       //disable gas inlet valves 
       //------------------------
       IF (#enb_prs_mon AND ("AV".ACT_PRS_GCH > "CNF".ACC_FNC_PRS_LIM)) THEN
           #dbl_gas_valves    :=  true;
       END_IF;
END_FUNCTION_BLOCK

FUNCTION_BLOCK "BM_MLT_GAP_SEARCH"   // FB117, SCL
{ S7_Optimized_Access := 'FALSE' }
VERSION : 0.0
// --------------------------------------------------------------------------------
//     program     :    BM_MLT_GAP_SEARCH
//     description :    melt gap search
//                          
//     name        :    G. Eibelshaeuser
//     date        :    19.10.2020
// 
//     revision    :
//     name        :
//     date        :    
//                     (c)PVA CGS GmbH
// --------------------------------------------------------------------------------
   VAR
      do_mlt_gap_search : Bool;
      mlt_gap_search_busy : Bool;
      "step" : Int;
      dly : Int;
      start_pos_xt : Real;
      start_pos_cr : Real;
   END_VAR
   VAR CONSTANT
      max_lft_dst : Real := 20.0;   // max lifting distance of crucible or crystal lift in [mm]
   END_VAR
BEGIN


       //disable melt gap search
       //-----------------------
       IF ("STA".ACT_STATE <> "APC".STATE_SERV) OR NOT ("LT".CR_LFT_UP XOR "LT".XT_LFT_DN) OR "LT".LSR_SEN_PWR_ON THEN
           "LT".MLT_GAP_SEARCH   :=  FALSE;
       //enable melt gap search
       //----------------------
       ELSE
           "SM_NEG_EDGE"(input   :=  "KYD".MLT_GAP_SEARCH,
                       busy    :=  #mlt_gap_search_busy,
                       output  :=  "LT".MLT_GAP_SEARCH);
       END_IF;

       //set activation flag melt gap search
       //-----------------------------------
       IF "LT".MLT_GAP_SEARCH THEN
           #do_mlt_gap_search   :=  true;
       END_IF;

       //melt gap search activated
       //-------------------------
       IF #do_mlt_gap_search THEN
           //abort melt gap search
           //---------------------
           IF NOT "LT".MLT_GAP_SEARCH THEN
               #step    :=  50;
           END_IF;

           //sequence
           //--------
           CASE #step OF 

               //switch on melt contact control
               //------------------------------
               0:  "KYD".MCC_ON  :=  TRUE;
                   //set speed set point
                   //-------------------
                   IF "LT".XT_LFT_DN THEN
                       "KYA".SET_XT_SPD  :=  1.0;
                   ELSIF "LT".CR_LFT_UP THEN
                       "KYA".SET_CR_SPD  :=  1.0;
                   END_IF;

                   //activate next step
                   //------------------
                   #step    :=  #step + 10;

               //store start position
               //--------------------
               10: #start_pos_xt    :=  "AV".ACT_XT_POS;
                   #start_pos_cr    :=  "AV".ACT_CR_POS;
                   #dly             :=  0;

                   //activate next step
                   //------------------
                   #step    :=  #step + 10;

               //find contact
               //------------    
               20: //crucible lift moved max. valid distance
                   //---------------------------------------
                   IF ("AV".ACT_CR_POS >= (#start_pos_cr + #max_lft_dst)) THEN
                       "KYD".CR_LFT_OFF          :=  TRUE;
                       "FLT".MLT_GAP_NO_CONTACT  :=  TRUE;
                   //crystal lift moved max. valid distance
                   //-------------------------------------
                   ELSIF ("AV".ACT_XT_POS >= (#start_pos_xt + #max_lft_dst)) THEN
                       "KYD".XT_LFT_OFF          :=  TRUE;
                       "FLT".MLT_GAP_NO_CONTACT  :=  TRUE;
                   //contact detected
                   //----------------
                   ELSIF "PDI".MCC_CONTACT_XT THEN
                       //stop crystal lift
                       //-----------------
                       IF  "LT".XT_LFT_DN THEN
                           "KYD".XT_LFT_OFF  :=  TRUE;
                           //activate next step
                           //------------------
                           #step    :=  #step + 10;
                       //stop crucible lift
                       //-----------------
                       ELSIF  "LT".CR_LFT_UP THEN   
                           "KYD".CR_LFT_OFF  :=  TRUE; 
                           //activate next step
                           //------------------
                           #step    :=  #step + 20;
                       END_IF;
                   END_IF;         

               //crystal - calculate distance
               //----------------------------
               30: IF NOT "LT".XT_LFT_DN THEN
                       //delay next step
                       //---------------
                       IF (#dly > 20) THEN
                           //calculate distance from contact to seed reference position
                           //---------------------------------------------------------- 
                           IF ("DIS".ACT_SEED_LSR_REF_POS > 0.0) THEN
                               "PAR_MAIN".MCONST_DST_LSR_MLT_LVL :=  "AV".ACT_XT_POS - "DIS".ACT_SEED_LSR_REF_POS;
                           END_IF;
                           //activate next step
                           //------------------
                           #step    :=  #step + 20;
                       ELSE
                           IF "SysTick100ms" THEN
                               #dly :=  #dly + 1;
                           END_IF;
                       END_IF;
                   END_IF;

               //crucible - store actual position
               //--------------------------------
               40: IF NOT "LT".CR_LFT_UP THEN
                       //delay next step
                       //---------------
                       IF (#dly > 20) THEN
                           //store actual crucible as dipping position
                           //----------------------------------------- 
                           "DIS".ACT_CR_DIP_POS  := "AV".ACT_CR_POS; 
                           //activate next step
                           //------------------
                           #step    :=  #step + 10;
                       ELSE
                           IF "SysTick100ms" THEN
                               #dly :=  #dly + 1;
                           END_IF;
                       END_IF;
                   END_IF;

               //reset off variables
               //-------------------
               50: "KYD".XT_LFT_OFF      :=  FALSE;
                   "KYD".CR_LFT_OFF      :=  FALSE;
                   "KYA".SET_XT_SPD      :=  0.0;
                   "KYA".SET_CR_SPD      :=  0.0;
                   #do_mlt_gap_search   :=  false;

           END_CASE;

       ELSE
           #step    :=  0;
           "FLT".MLT_GAP_NO_CONTACT  :=  FALSE;
       END_IF;
END_FUNCTION_BLOCK

FUNCTION_BLOCK "BM_SEED_REF_POS"   // FB118, SCL
{ S7_Optimized_Access := 'FALSE' }
VERSION : 0.0
// --------------------------------------------------------------------------------
//     program     :    BM_SEED_REF_POS
//     description :    seed reference position search
//                          
//     name        :    G. Eibelshaeuser
//     date        :    18.12.2020
// 
//     revision    :
//     name        :
//     date        :    
//                     (c)PVA CGS GmbH
// --------------------------------------------------------------------------------
   VAR
      do_ref_search : Bool;
      seed_search_busy : Bool;
      lsr_sen_obj_det : Bool;
      "step" : Int;
      dly : Int;
      start_pos_xt : Real;
   END_VAR
   VAR CONSTANT
      max_lft_dst : Real := 20.0;   // max lifting distance of crucible or crystal lift in [mm]
   END_VAR
BEGIN


       //switch on laser in dipping phase
       //--------------------------------
       IF ("APC".STATUS = "APC".DIPPING) THEN
           "LT".LSR_SEN_PWR_ON   :=  TRUE;        
       //disable reference search
       //------------------------
       ELSIF "APC".AUTOMATIC OR NOT "LT".XT_LFT_DN OR "LT".MLT_GAP_SEARCH THEN
           "LT".LSR_SEN_PWR_ON   :=  FALSE;
       //enablereference search
       //----------------------
       ELSE
           "SM_NEG_EDGE"(input   :=  "KYD".LSR_SEN_PWR_ON,
                       busy    :=  #seed_search_busy,
                       output  :=  "LT".LSR_SEN_PWR_ON);
       END_IF;

       //set activation flag melt gap search
       //-----------------------------------
       IF ("LT".LSR_SEN_PWR_ON AND ("APC".STATUS = "APC".IDLE))THEN
           #do_ref_search   :=  true;
       END_IF;

       //reference search activated
       //--------------------------
       IF #do_ref_search THEN
           //abort reference position search
           //-------------------------------
           IF (NOT "LT".LSR_SEN_PWR_ON AND (#step < 25)) THEN
               #step    :=  40;
           END_IF;

           //sequence
           //--------
           CASE #step OF 
               //switch on melt contact control
               //------------------------------
               0:  //set speed set point
                   //-------------------
                   "KYA".SET_XT_SPD              :=  1.0;
                   "DIS".ACT_SEED_LSR_REF_POS    :=  0.0;
                   #dly                         :=  0;
                   //activate next step
                   //------------------
                   #step    :=  #step + 10;

               //store start position
               //--------------------
               10: #start_pos_xt    :=  "AV".ACT_XT_POS;
                   //activate next step
                   //------------------
                   #step    :=  #step + 10;

               //find contact
               //------------    
               20: //crystal lift moved max. valid distance
                   //-------------------------------------
                   IF ("AV".ACT_XT_POS >= (#start_pos_xt + #max_lft_dst)) THEN
                       "KYD".XT_LFT_OFF  :=  TRUE;
                       //activate next step
                       //------------------
                       #step    :=  #step + 5;
                   //reference position detected with positive edge of laser sensor
                   //--------------------------------------------------------------
                   ELSIF ("PDI".LSR_SEN_OBJ_DET AND NOT #lsr_sen_obj_det) THEN
                       "KYD".XT_LFT_OFF  :=  TRUE;
                       //activate next step
                       //------------------
                       #step    :=  #step + 10;
                   END_IF;

               25: //crystal lift stopped - no seed detected within valid range
                   //----------------------------------------------------------
                   IF NOT "LT".XT_LFT_DN THEN
                       "FLT".SEED_DET    :=  TRUE;
                       //delay next step
                       //---------------
                       IF (#dly > 20) THEN 
                           //activate next step
                           //------------------
                           #step    :=  #step + 15;
                       ELSE
                           IF "SysTick100ms" THEN
                               #dly :=  #dly + 1;
                           END_IF;
                       END_IF;
                   END_IF;

               30: //crystal lift stopped - position stored
                   //--------------------------------------
                   IF NOT "LT".XT_LFT_DN THEN
                       //delay next step
                       //---------------
                       IF (#dly > 20) THEN 
                           //store actual position as reference position
                           //-------------------------------------------
                           "DIS".ACT_SEED_LSR_REF_POS    :=  "AV".ACT_XT_POS;
                           //activate next step
                           //------------------
                           #step    :=  #step + 10;
                       ELSE
                           IF "SysTick100ms" THEN
                               #dly :=  #dly + 1;
                           END_IF;
                       END_IF;

                   END_IF;

               //reset off variables
               //-------------------
               40: "KYD".XT_LFT_OFF      :=  FALSE;
                   "KYA".SET_XT_SPD      :=  0.0;
                   "LT".LSR_SEN_PWR_ON   :=  FALSE;
                   #do_ref_search       :=  false;

           END_CASE;

       ELSE
           #step            :=  0;
           "FLT".SEED_DET    :=  FALSE;
       END_IF;

       //store status of current cycle
       //-----------------------------
       #lsr_sen_obj_det :=  "PDI".LSR_SEN_OBJ_DET;

       //set output laser power on
       //-------------------------
       "PDO".LSR_SEN_PWR_ON  :=  NOT "LT".LSR_SEN_PWR_ON;  //output must be "false" for laser on!!!
END_FUNCTION_BLOCK

FUNCTION_BLOCK "CM_PT1"   // FB130, SCL
{ S7_Optimized_Access := 'FALSE' }
VERSION : 0.0
// --------------------------------------------------------------------------------
//     program     :    CM_PT1
//     description :    pt1 filter 
//     name        :    K. Kalkowski
//     date        :    29.10.99
// 
//     revision    :    1.00
//     name        :    K. Kalkowski
//     date        :    29.10.99
// 
//                     (c)LEYBOLD SYSTEMS
//     --------------------------------------------------------------------------------
   VAR_INPUT
      u_in : Real;   // filter input
      t1_in : Real;   // filter time in sec.
      ts_in : Real;   // filter sample time
      tc_in : Real;   // interrupt time for filter module call (ts/tc>=1, ts/tc=integer!)
      range_in : Real;   // value for 100% input (e.g. 8mm/min = 100%) used for u_in
      range_out : Real;   // value for 100% output (e.g. 700C = 100%) used for y_out
      y_llim : Real;   // low limit for y_out
      y_hlim : Real;   // high limit for y_out
   END_VAR
   VAR_IN_OUT
      y_out : Real;   // pt1 filter output
   END_VAR
   VAR
      u : Real;   // filter input
      y_sum : Real;   // sum of pt1 components
      filter_call_cycle : Int;   // pt1 algorithm call every (ts/tc) cycles
      hlim_active : Bool;   // hlim active
      llim_active : Bool;   // llim active
      filter_off : Bool;   // filter function off (T1 = 0)
      ctrl_call_cycle : Int;   // pt1 algorithm call every (ts/tc) cycles
   END_VAR
BEGIN


       IF #range_in = 0 THEN                                            //check range_in value
           #u:= 0;
       ELSE
           #u:= #u_in / #range_in;
       END_IF;

       IF  #ctrl_call_cycle >= REAL_TO_INT(#ts_in/#tc_in)THEN             //wait for next controller call                               
           #ctrl_call_cycle := 1;
           IF #t1_in <= 0.0 THEN
               #filter_off := true;      
           ELSE
               #filter_off := false;      
           END_IF;
           IF #filter_off = false THEN
               ENO:=TRUE;
               #y_sum := #y_sum + (#u - #y_sum) * (#ts_in/#t1_in);           //calculate filter function
               IF ENO = FALSE THEN
                   #y_sum:=0.0;
               END_IF; 
           ELSE
               #y_sum := #u;
           END_IF;
       ELSE    
           #ctrl_call_cycle := #ctrl_call_cycle + 1;
       END_IF;

       IF #y_sum > #y_hlim / #range_out THEN                              //limit and convert output
           #y_sum := #y_hlim / #range_out;
           #hlim_active := true;
       ELSE
           #hlim_active := false;
       END_IF;
       IF #y_sum < #y_llim / #range_out THEN
           #y_sum := #y_llim / #range_out;
           #llim_active := true;     
       ELSE
           #llim_active := false;
       END_IF;                                                              
       #y_out := #y_sum * #range_out;                                     //set output value
END_FUNCTION_BLOCK

FUNCTION_BLOCK "CM_PT2"   // FB131, SCL
{ S7_Optimized_Access := 'FALSE' }
VERSION : 0.0
// --------------------------------------------------------------------------------
//     program     :    CM_PT2
//     description :    pt2 filter 
//     name        :    G. Eibelsh鋟ser
//     date        :    20.02.2001
// 
//     revision    :    
//     name        :    
//     date        :    
// 
//                     (c)CGS
//     --------------------------------------------------------------------------------
   VAR_INPUT
      u_in : Real;   // filter input
      t1_in : Real;   // filter time 1 in sec.
      t2_in : Real;   // filter time 2 in sec.
      ts_in : Real;   // filter sample time
      tc_in : Real;   // interrupt time for filter module call (ts/tc>=1, ts/tc=integer!)
      range_in : Real;   // value for 100% input (e.g. 8mm/min = 100%) used for u_in
      range_out : Real;   // value for 100% output (e.g. 700C = 100%) used for y_out
      y_llim : Real;   // low limit for y_out
      y_hlim : Real;   // high limit for y_out
   END_VAR
   VAR_IN_OUT
      y_out : Real;   // pt2 filter output
   END_VAR
   VAR
      u : Real;   // filter input
      y_sum : Real;   // sum of pt2 components
      filter_call_cycle : Int;   // pt2 algorithm call every (ts/tc) cycles
      hlim_active : Bool;   // hlim active
      llim_active : Bool;   // llim active
      filter_off : Bool;   // filter function off (T1 = 0)
      ctrl_call_cycle : Int;   // pt2 algorithm call every (ts/tc) cycles
   END_VAR
BEGIN


       IF #range_in = 0 THEN                                            //check range_in value
           #u:= 0;
       ELSE
           #u:= #u_in / #range_in;
       END_IF;

       IF  #ctrl_call_cycle >= REAL_TO_INT(#ts_in/#tc_in)THEN             //wait for next controller call                               
           #ctrl_call_cycle := 1;

           IF (#t1_in <= 0.0)  THEN
               #filter_off := true;      
           ELSE
               #filter_off := false;      
           END_IF;

           IF #filter_off = false THEN
               ENO:= TRUE;
               #y_sum := #y_sum + (#u - #y_sum) * #ts_in/(1+#t1_in+#t2_in+#t1_in*#t2_in);   //calculate filter function
               IF ENO = FALSE THEN
                   #y_sum:=0.0;
               END_IF; 
           ELSE
               #y_sum := #u;
           END_IF;
       ELSE    
           #ctrl_call_cycle := #ctrl_call_cycle + 1;
       END_IF;

       IF #y_sum > #y_hlim / #range_out THEN                              //limit and convert output
           #y_sum := #y_hlim / #range_out;
           #hlim_active := true;
       ELSE
           #hlim_active := false;
       END_IF;
       IF #y_sum < #y_llim / #range_out THEN
           #y_sum := #y_llim / #range_out;
           #llim_active := true;     
       ELSE
           #llim_active := false;
       END_IF;                                                              
       #y_out := #y_sum * #range_out;                                     //set output value
END_FUNCTION_BLOCK

FUNCTION_BLOCK "CM_DT1"   // FB132, SCL
{ S7_Optimized_Access := 'FALSE' }
VERSION : 0.0
// --------------------------------------------------------------------------------
//     program     :    CM_DT1
//     description :    dt1 derivative function with delay 
//     name        :    K. Kalkowski
//     date        :    26.11.99
// 
//     revision    :    1.00
//     name        :    K. Kalkowski
//     date        :    26.11.99
// 
//                     (c)LEYBOLD SYSTEMS
//     --------------------------------------------------------------------------------
   VAR_INPUT
      u_in : Real;   // function input
      td_in : Real;   // derivative time const. in sec.
      t1_in : Real;   // derivative delay time in sec.
      ts_in : Real;   // function sample time
      tc_in : Real;   // interrupt time for function module call (ts/tc>=1, ts/tc=integer!)
      range_in : Real;   // value for 100% input (e.g. 8mm/min = 100%) used for u_in
      range_out : Real;   // value for 100% output (e.g. 700C = 100%) used for y_out
      y_llim : Real;   // low limit for y_out
      y_hlim : Real;   // high limit for y_out
   END_VAR
   VAR_IN_OUT
      y_out : Real;   // dt1 function output
   END_VAR
   VAR
      u : Real;   // function input
      u_old : Real;   // previous of u
      y_sum : Real;   // sum of dt1 components
      funct_call_cycle : Int;   // dt1 algorithm call every (ts/tc) cycles
      hlim_active : Bool;   // hlim active
      llim_active : Bool;   // llim active
      funct_off : Bool;   // dt1 function off (Td = 0)
      ctrl_call_cycle : Int;   // dt1 algorithm call every (ts/tc) cycles
      xd : Real;   // set - act
      xd_old : Real;   // previous value of xd
      du : Real;   // u - u_old
      dxr : Real;   // xr n (differenzenquotient)
      dxr_old : Real;   // xr,n-1 (previous differenzenquotient)
   END_VAR
BEGIN


       IF #range_in = 0 THEN                                        //check range_in value
           #u:= 0;
       ELSE
           #u:= #u_in / #range_in;
           //dxr := 0;
       END_IF;

       IF  #ctrl_call_cycle >= REAL_TO_INT(#ts_in/#tc_in)THEN         //wait for next controller call                               
           #ctrl_call_cycle := 1;
           #du := #u - #u_old;                                        //calculate input                                         
           IF #td_in <= 0.0 THEN
               #funct_off := true;      
           ELSE
               #funct_off := false;      
           END_IF;
           IF #funct_off = false THEN                               //calculate dt1 function
               ENO:=TRUE;
               #dxr := (#du + (#t1_in * #dxr_old)) / (#ts_in + #t1_in);  //differenzenquotient
               IF ENO = FALSE THEN
                   #dxr_old:=0.0;
                   #dxr:=0.0;
               END_IF;              
               #y_sum := #td_in * #dxr;                               //dt1    
           ELSE
               #y_sum := #u;
           END_IF;
           #u_old := #u;                                                 //save previous values
           #dxr_old := #dxr;
       ELSE    
           #ctrl_call_cycle := #ctrl_call_cycle + 1;
       END_IF;

       IF #y_sum > #y_hlim / #range_out THEN                          //limit and convert output
           #y_sum := #y_hlim / #range_out;
           #hlim_active := true;
       ELSE
           #hlim_active := false;
       END_IF;
       IF #y_sum < #y_llim / #range_out THEN
           #y_sum := #y_llim / #range_out;
           #llim_active := true;     
       ELSE
           #llim_active := false;
       END_IF;                                                              
       #y_out := #y_sum * #range_out;                                 //set output value
END_FUNCTION_BLOCK

FUNCTION_BLOCK "CM_INC"   // FB133, SCL
{ S7_Optimized_Access := 'FALSE' }
VERSION : 0.0
// --------------------------------------------------------------------------------
//     program     :    CM_INC
//     description :    increment function  
//     name        :    K. Kalkowski
//     date        :    26.11.99
// 
//     revision    :    1.00
//     name        :    K. Kalkowski
//     date        :    26.11.99
//     
//     revision    :    minimum increment limit added
//     name        :    G. Eibelsh鋟ser
//     date        :    28.11.2011
// 
//                     (c)PVA TePla AG
//     --------------------------------------------------------------------------------
   VAR_INPUT
      u1_in : Real;   // increment input 1
      u2_in : Real;   // increment input 2
      u3_in : Real;   // increment input 3
      k1_in : Real;   // factor for increment input 1
      k2_in : Real;   // factor for increment input 2
      k3_in : Real;   // factor for increment input 3
      y0_in : Real;   // start value input
      y_llim : Real;   // low limit for y_out
      y_hlim : Real;   // high limit for y_out
      y0_mode : Bool;   // set start value of increment function
   END_VAR
   VAR_IN_OUT
      y_out : Real;   // inc function output
      stp_1 : Bool;   // stop increment function (used for change of input connection)
      stp_2 : Bool;
      stp_3 : Bool;
      rstrt_1 : Bool;   // restart increment function (used for start of new increment table)
      rstrt_2 : Bool;
      rstrt_3 : Bool;
   END_VAR
   VAR
      u1_old : Real;   // increment 1 input of previous call
      u2_old : Real;   // increment 2 input of previous call
      u3_old : Real;   // increment 3 input of previous call
      y0 : Real;   // start value
      y_sum : Real;   // sum of increments
      stp1_i : Int;   // index stop function
      stp2_i : Int;
      stp3_i : Int;
      rstrt1_i : Int;   // index restart function
      rstrt2_i : Int;
      rstrt3_i : Int;
   END_VAR
   VAR CONSTANT
      min_inc : Real := 0.001;
   END_VAR
BEGIN


       IF #stp_1 THEN                                    //stop inc function
           #stp1_i := #stp1_i + 1;
           IF (#stp1_i > 2) THEN
               #stp_1 := false;
           END_IF;    
       ELSE
           #stp1_i := 0;
       END_IF;    

       IF #stp_2 THEN
           #stp2_i := #stp2_i + 1;
           IF (#stp2_i > 2) THEN
               #stp_2 := false;
           END_IF;    
       ELSE
           #stp2_i := 0;
       END_IF;    

       IF #stp_3 THEN
           #stp3_i := #stp3_i + 1;
           IF (#stp3_i > 2) THEN
               #stp_3 := false;
           END_IF;    
       ELSE
           #stp3_i := 0;
       END_IF;    

       IF #rstrt_1 THEN                                  //restart inc function
           #rstrt1_i := #rstrt1_i + 1;
           IF (#rstrt1_i > 2) THEN
               #rstrt_1 := false;
           END_IF;    
       ELSE
           #rstrt1_i := 0;
       END_IF;    

       IF #rstrt_2 THEN                                    
           #rstrt2_i := #rstrt2_i + 1;
           IF (#rstrt2_i > 2) THEN
               #rstrt_2 := false;
           END_IF;    
       ELSE
           #rstrt2_i := 0;
       END_IF;    

       IF #rstrt_3 THEN                                    
           #rstrt3_i := #rstrt3_i + 1;
           IF (#rstrt3_i > 2) THEN
               #rstrt_3 := false;
           END_IF;    
       ELSE
           #rstrt3_i := 0;
       END_IF;    

       IF NOT #y0_mode THEN                                         //calculate y_sum
           IF NOT (#rstrt_1 OR #stp_1) THEN 
               IF (ABS(#u1_in - #u1_old) >= #min_inc) THEN            //check if increment is larger than minimum increment limit           
                   #y_sum   := #y_sum + ((#u1_in - #u1_old)*#k1_in);
                   #u1_old  := #u1_in;                               //store last input value
               END_IF;
           END_IF;

           IF NOT (#rstrt_2 OR #stp_2) THEN
               IF (ABS(#u2_in - #u2_old) >= #min_inc) THEN                  
                   #y_sum   := #y_sum + ((#u2_in - #u2_old)*#k2_in);
                   #u2_old  := #u2_in;
               END_IF;
           END_IF;

           IF NOT (#rstrt_3 OR #stp_3) THEN
               IF (ABS(#u3_in - #u3_old) >= #min_inc) THEN                  
                   #y_sum   := #y_sum + ((#u3_in - #u3_old)*#k3_in);
                   #u3_old  := #u3_in;
               END_IF;
           END_IF;

       ELSE
           #y_sum   := #y0_in;
           #u1_old  := #u1_in;
           #u2_old  := #u2_in;
           #u3_old  := #u3_in;

       END_IF;

       IF #y_sum > #y_hlim THEN                                  //limit y_sum
           #y_sum := #y_hlim;    
       END_IF;
       IF #y_sum < #y_llim THEN
           #y_sum := #y_llim;    
       END_IF;

       IF #rstrt_1 THEN                                         //reset previous values
           #u1_old := 0.0;
       END_IF;

       IF #stp_1 THEN
           #u1_old := #u1_in;
       END_IF;

       IF #rstrt_2 THEN
           #u2_old := 0.0;
       END_IF;

       IF #stp_2 THEN
           #u2_old := #u2_in;
       END_IF;

       IF #rstrt_3 THEN
           #u3_old := 0.0;
       END_IF;

       IF #stp_3 THEN
           #u3_old := #u3_in;
       END_IF;

       #y_out := #y_sum;                                         //set output
END_FUNCTION_BLOCK

FUNCTION_BLOCK "CM_LOOP_PRS"   // FB134, SCL
{ S7_Optimized_Access := 'FALSE' }
VERSION : 0.0
// --------------------------------------------------------------------------------
//     program     :    CM_LOOP_PRS
//     description :    pressure control loop 
//     name        :    K. Kalkowski
//     date        :    07.12.99
// 
//     revision    :    call of CONT_C added as alternative
//     name        :    G. Eibelsh鋟ser
//     date        :    06.09.2007
//    
//     revision    :    
//     name        :    
//     date        :    
// 
//                     (c)PVA TePla AG
//     --------------------------------------------------------------------------------
   VAR
      STD_PID : CONT_C;   // standard Siemens controller algorithm
      PT1 : "CM_PT1";   // pt1 filter for actual xtal diameter
      ramp_enb : Bool;
      cyc_cnt : Bool;
      int_hold_req : Bool;   // integral hold action request
      ctl_prs_on : Bool;
      cycle : Int;
      count : Int;
      ctrl_calls : Int;   // controller call counter
      set : Real;   // internal set point
      act : Real;   // internal actual value
      hand : Real;   // internal hand value
      set_ramp : Real;
   END_VAR
   VAR_TEMP
      high_lim_active : Bool;   // high limit of controller output is reached
      low_lim_active : Bool;   // low limit of controller output is reached
      int_action_on : Bool;   // integral action on
      der_action_on : Bool;   // derivative action on
      per_out : Word;   // peripherial controller output variable
      p_part_out : Real;   // proportionality component
      i_part_out : Real;   // integral component
      d_part_out : Real;   // derivative component
      eff_act_val : Real;   // effective process variable
      error_sig : Real;   // control deviation
   END_VAR
   VAR CONSTANT
      nc : Real := 0.0;   // "not connected input"
   END_VAR
BEGIN


       //build hand value
       //---------------- 
       #hand := "CM_INSELECT" (auto   := ("APC".AUTOMATIC AND NOT "SY".CTL_PRS_SMI) OR "DV".SI_FIL_FSH_SEQ_ON,        
                            track  := false,
                            ac     := "AC".SET_CTL_VALVE_POS,                
                            kya    := "KYA".SET_CTL_VALVE_POS);                    

       //build set point
       //---------------
       #set := "CM_INSELECT"(auto    := "APC".AUTOMATIC AND NOT "SY".CTL_PRS_SMI,            
                          track   := true,
                          ac      := "AC".SET_CLF_PRS,
                          kya     := "KYA".SET_PRS_FNC);

       //limitation of pressure control setpoint if no 1000mbar Baratron on furnace chamber present
       //-----------------------------------------------------------------------------------------                   
       IF NOT "CNF".CONF_CLF_BAR_1000    THEN        // check config flag
           IF #set > 90.0 THEN                      // pressure control setpoint limited to 90 mbar
               #set             := 90.0;
               "KYA".SET_PRS_FNC := #set;       
           END_IF;
       END_IF;                    

       #act := "AV".ACT_PRS_FCH;                              //read actual value

       //built controller on flag
       //------------------------
       IF "DV".SI_FIL_FSH_SEQ_ON OR NOT "PDI".EMO THEN 
           "SY".CTL_PRS_ON := FALSE;                 
       ELSIF "DV".FIL_CLN_REQ_IN_PRC THEN        //prevent switch off of pressure control when filter cleaning during process is active
           "SY".CTL_PRS_ON := TRUE;                 
       ELSIF "APC".AUTOMATIC THEN  
           "SY".CTL_PRS_ON := "DC".CTL_PRS_ON;                 
       ELSE 
           "SY".CTL_PRS_ON := ("SY".CTL_PRS_ON AND NOT "KYD".CTL_PRS_OFF) OR "KYD".CTL_PRS_ON; 
       END_IF;

       //setpoint ramping
       //----------------
       IF "SY".CTL_PRS_ON    THEN
           // call setpoint ramp function after controller start
           //---------------------------------------------------
           IF ("PAR_SUB".PRS_RP_GRAD > 0.0)     THEN
               "CM_SET_RAMP"(rp_enb      := #ramp_enb,
                           i           := #cyc_cnt,
                           max_dev     := "PAR_SUB".PRS_RP_MAX_DEV,
                           rp_start    := "PAR_SUB".PRS_RP_START,
                           rp_grad     := "PAR_SUB".PRS_RP_GRAD,
                           tme_base    := 60.0,
                           tc_in       := 0.1,
                           set_p       := #set,
                           act_v       := #act,
                           set_out     := #set_ramp);

               #set     := #set_ramp; 
           END_IF;  
       ELSE
           #ramp_enb  := TRUE;     
           #cyc_cnt   := TRUE;                
       END_IF;

       //write setpoint in KYA variable 
       //------------------------------
       IF "APC".AUTOMATIC AND NOT "SY".CTL_PRS_SMI THEN   
           "KYA".SET_PRS_FNC := #set;
       END_IF;

       "LT".CTL_PRS_ON := "SY".CTL_PRS_ON;                             

       //chose parameter set according to pressure setpoint
       //--------------------------------------------------
       IF #set <= 100.0 THEN
           "AC".CTL_PRS_GN := "PAR_MAIN".CTL_PRS_GN;               //fetch pid parameter from par_main db
           "AC".CTL_PRS_TI := "PAR_MAIN".CTL_PRS_TI;
           "AC".CTL_PRS_TD := "PAR_MAIN".CTL_PRS_TD;
           "AC".CTL_PRS_T1 := "PAR_MAIN".CTL_PRS_T1;    
       ELSE
           "AC".CTL_PRS_GN := "PAR_MAIN".CTL_PRS_GN_HI;               //fetch pid parameter from par_main db
           "AC".CTL_PRS_TI := "PAR_MAIN".CTL_PRS_TI_HI;
           "AC".CTL_PRS_TD := "PAR_MAIN".CTL_PRS_TD_HI;
           "AC".CTL_PRS_T1 := "PAR_MAIN".CTL_PRS_T1_HI;    
       END_IF;    

       //change polarity of control values
       //---------------------------------
       #set := #set *(-1);                                                          
       #act := #act *(-1);                                               

       //do controller call
       //------------------

           //switch off pressure controller
           //------------------------------ 
           IF NOT "SY".CTL_PRS_ON    THEN 
               #ctl_prs_on  :=  false;
           END_IF;

           //enable of single controller actions
           //----------------------------------- 
           IF ("AC".CTL_PRS_TI > 0.0)   THEN         //i- part
               #int_action_on   :=  true;
           ELSE
               #int_action_on   :=  false;
           END_IF;

           IF ("AC".CTL_PRS_TD > 0.0)   THEN         //d-part
               #der_action_on   :=  true;
           ELSE
               #der_action_on   :=  false;
           END_IF;

           //call Standard PID controller 
           //----------------------------
           #STD_PID(COM_RST         :=  "KYD".PRS_CTRL_RST,                   //restart of controller, resets controller values
                   MAN_ON          :=  NOT #ctl_prs_on,                     //switch controller on/off
                   PVPER_ON        :=  false,                              //activate reading of peripherie value
                   P_SEL           :=  true,                               //proportional action on
                   I_SEL           :=  #int_action_on,                      //integral action on
                   INT_HOLD        :=  #int_hold_req,                       //integral action hold
                   I_ITL_ON        :=  false,                              //initialization of the integral action - set value of I_ITLVAL
                   D_SEL           :=  #der_action_on,                      //derivative action on
                   CYCLE           :=  T#100ms,                            //sample time
                   SP_INT          :=  #set,                                //internal setpoint
                   PV_IN           :=  #act,                                //process variable input
                   PV_PER          :=  W#16#0000,                          //process variable peripherial input
                   MAN             :=  #hand,                               //hand value as percentaged input
                   GAIN            :=  "AC".CTL_PRS_GN,                      //controller gain
                   TI              :=  DINT_TO_TIME(REAL_TO_DINT("AC".CTL_PRS_TI * 1000.0)), //integration time
                   TD              :=  DINT_TO_TIME(REAL_TO_DINT("AC".CTL_PRS_TD * 1000.0)), //derivative time
                   TM_LAG          :=  DINT_TO_TIME(REAL_TO_DINT("AC".CTL_PRS_T1 * 1000.0)), //time lag of the derivative action
                   DEADB_W         :=  0.0,                            //dead band of control deviation
                   LMN_HLM         :=  100.0,                          //upper limit of controller output as percentaged value 
                   LMN_LLM         :=  0.0,                            //lower limit of controller output as percentaged value
                   PV_FAC          :=  1.0,                            //process variable factor (used on peripherial input)
                   PV_OFF          :=  0.0,                            //process variable offset
                   LMN_FAC         :=  1.0,                            //output standardization(percentage to physical value)
                   LMN_OFF         :=  0.0,                            //offset of output value
                   I_ITLVAL        :=  0.0,                            //initialization value of the integral action
                   DISV            :=  #nc);                            //disturbance variable

                   //write output variables of PID controller
                   //----------------------------------------
                   "CTL".SET_CTL_VALVE_POS  :=  #STD_PID.LMN;                 //controller output variable as physical value

                   #per_out         :=  #STD_PID.LMN_PER;                    //peripherial controller output variable
                   #high_lim_active :=  #STD_PID.QLMN_HLM;                   //high limit of controller output is reached
                   #low_lim_active  :=  #STD_PID.QLMN_LLM;                   //low limit of controller output is reached
                   #p_part_out      :=  #STD_PID.LMN_P;                      //proportionality component
                   #i_part_out      :=  #STD_PID.LMN_I;                      //integral component
                   #d_part_out      :=  #STD_PID.LMN_D;                      //derivative component
                   #eff_act_val     :=  #STD_PID.PV;                         //effective process variable 
                   #error_sig       :=  #STD_PID.ER;                         //control deviation

           //evaluate controller output limits
           //---------------------------------
           IF #high_lim_active XOR #low_lim_active   THEN                //check controller limits
               IF (#ctrl_calls > 50) THEN                                   
                   IF #high_lim_active AND (#i_part_out > 0.0)   THEN 
                       #int_hold_req    :=  true;                       //set integral action on hold
                   ELSIF #low_lim_active AND (#i_part_out < 0.0) THEN 
                       #int_hold_req    :=  true;                       //set integral action on hold
                   ELSE 
                       #int_hold_req    :=  false;                      //reset integral action on hold
                   END_IF;
               ELSE
                   #ctrl_calls  :=  #ctrl_calls + 1;                     //count controller calls
               END_IF;
           ELSE
               #ctrl_calls      :=  0;                                  //reset controller call counts
               #int_hold_req    :=  false;                              //reset integral action hold request
           END_IF;

           //switch on pressure controller
           //------------------------------ 
           IF "SY".CTL_PRS_ON    THEN 
               #ctl_prs_on  :=  true;
           END_IF;                

           //track KYA value of pressure control set point
           //---------------------------------------------
           IF (("APC".AUTOMATIC OR "SY".CTL_PRS_ON OR "DV".SI_FIL_FSH_SEQ_ON) AND NOT "DV".V1_HAND_MODE) THEN 
               "KYA".SET_CTL_VALVE_POS   :=  "CTL".SET_CTL_VALVE_POS;
           END_IF;
END_FUNCTION_BLOCK

FUNCTION_BLOCK "CM_LOOP_DIA"   // FB135, SCL
{ S7_Optimized_Access := 'FALSE' }
VERSION : 0.0
// --------------------------------------------------------------------------------
//     program     :    CM_LOOP_DIA
//     description :    xtal diameter control loop 
//     name        :    K. Kalkowski
//     date        :    02.12.99
// 
//     revision    :    call of CONT_C added as alternative
//     name        :    G. Eibelsh鋟ser
//     date        :    29.08.2007
//    
//     revision    :    
//     name        :    
//     date        :    
// 
//                     (c)PVA TePla AG
//     --------------------------------------------------------------------------------
   VAR
      STD_PID : CONT_C;   // standard Siemens controller algorithm
      PT2 : "CM_PT2";   // pt2 filter for xtal diameter
      DYN_WIN : "CM_DYN_WIN";   // filter to eliminate spurious measurements
      int_hold_req : Bool;   // integral hold action request
      ramp_enb : Bool;
      cyc_cnt : Bool;
      ctl_dia_on : Bool;
      ne_dia_ctrl_off : Bool;
      xt_spd_chg_done : Bool;
      add_spd_inc : Bool;
      dia_below_lim : Bool;
      dia_below_lim_old : Bool;
      cycle : Int;
      count : Int;
      ctrl_calls : Int;   // controller call counter
      i : Int;
      ctrl_calls_gap : Int;
      ctrl_calls_speed : Int;
      set : Real;   // internal set point
      act : Real;   // internal actual value
      hand : Real;   // hand value
      hand_int : Real;   // internal hand value (only used for CONT_C algorithm)
      ll : Real;   // internal low_lim xt - speed
      hl : Real;   // internal hi_lim xt - speed
      set_ramp : Real;
      dia_prev_call : Real;
      delta_prev_call : Real;
      set_prv_cyc : Real;
      hand_gap : Real;
   END_VAR
   VAR_TEMP
      set_enable : Bool;   // enable signal for filter function
      high_lim_active : Bool;   // high limit of controller output is reached
      low_lim_active : Bool;   // low limit of controller output is reached
      int_action_on : Bool;   // integral action on
      der_action_on : Bool;   // derivative action on
      per_out : Word;   // peripherial controller output variable
      p_part_out : Real;   // proportionality component
      i_part_out : Real;   // integral component
      d_part_out : Real;   // derivative component
      eff_act_val : Real;   // effective process variable
      error_sig : Real;   // control deviation
   END_VAR
   VAR CONSTANT
      nc : Real := 0.0;   // "not connected input"
   END_VAR
BEGIN


       //neck phase active and speed increment at lowest diameter requested
       //------------------------------------------------------------------
       IF (("APC".STATUS = "APC".NECK) AND ("PAR_MAIN".NE_MIN_DIA >= 0.1) AND (ABS("PAR_MAIN".NE_XT_SPD_INC) >= 0.1)) THEN    

           //reset neck diameter below limit flag after 60sec.
           //-------------------------------------------------
           IF (#i >= 600) THEN
               #dia_below_lim   :=  false;
               #i               :=  0;
           //increase counter every 100ms if neck diameter below limit flag is set
           //---------------------------------------------------------------------
           ELSIF #dia_below_lim THEN
               #i := #i + 1;
           //set neck diameter below limit flag
           //----------------------------------
           ELSIF (("AV".ACT_XT_DIA < "PAR_MAIN".NE_MIN_DIA) AND "SY".CTL_DIA_ON AND "DV".CAM_ISP_ON) THEN
               #dia_below_lim   :=  true;
           END_IF;

           //detect positive edge of "neck diameter below limit" fault
           //---------------------------------------------------------
           IF #dia_below_lim AND NOT #dia_below_lim_old THEN
               #add_spd_inc := true;
           END_IF;

           //built control off flag when neck diameter reached minimum diameter
           //------------------------------------------------------------------
           IF #xt_spd_chg_done THEN                         //crystal speed change done
               #ne_dia_ctrl_off := false;                   //reset controller off variable - restart controller again    
               #xt_spd_chg_done := false;                   //reset speed change done status

           //neck diameter at minimum diameter
           //---------------------------------
           ELSIF #add_spd_inc THEN
               #ne_dia_ctrl_off := true;                    //switch off diameter controller 

               //controller is off - add increment to manual set point
               //-----------------------------------------------------
               IF NOT #ctl_dia_on THEN
                   "KYA".SET_XT_SPD  := "KYA".SET_XT_SPD + "PAR_MAIN".NE_XT_SPD_INC; //add crystal speed increment to manual set point

                   //limit lowest speed set point with recipe value
                   //----------------------------------------------
                   IF ("KYA".SET_XT_SPD < "AC".SET_XT_SPD_DEV_2) THEN
                       "KYA".SET_XT_SPD  := "AC".SET_XT_SPD_DEV_2;
                   END_IF;

                   #xt_spd_chg_done := true;            //set speed change done status
                   #add_spd_inc     := false;           //reset add speed increment variable
               END_IF;
           END_IF;

           //store status of neck diameter below limit fault
           //-----------------------------------------------
           #dia_below_lim_old := #dia_below_lim;  

       ELSE
           #ne_dia_ctrl_off     := false;           //reset controller off variable
           #xt_spd_chg_done     := false;           //reset speed change done status
           #add_spd_inc         := false;           //reset add speed increment variable
           #dia_below_lim       := false;           //reset neck diameter below limit flag
           #dia_below_lim_old   := false;           //reset neck diameter limit flag of previous cycle
           #i                   := 0;               //reset counter
       END_IF;

       //build hand value 
       //----------------
       IF ("CTL".SET_SPEED_OFFS = 0.0) THEN  //offset speed controller off and output ramped down to zero
           #hand := "CM_INSELECT" (auto   := ("APC".AUTOMATIC AND NOT "SY".CTL_DIA_SMI AND NOT #ne_dia_ctrl_off),      //hand value used when dia controller is off    
                                track  := false,
                                ac     := "AC".SET_XT_SPD,                
                                kya    := "KYA".SET_XT_SPD); 
       ELSE
           #hand := "CTL".SET_XT_SPD; //keep dia controller output as hand value as long as output of offset speed controller is ramp down to zero
       END_IF;


       //read setpoint
       //-------------
       #set := "AC".SET_XT_DIA;                           

       //set_enable  :=   BM_CAM_CONTROL_DB.CAM_DIA   AND (APC.STATUS <> 4);     //STATUS 4 = DIPPING

       //call dynamic measurement window
       //-------------------------------              
       #DYN_WIN (enb            := false, //set_enable,             //enable signal for filter function 
                u_in           := "AV".INP_XT_DIA,                   //actual diameter value from width analyser  
                t1_in          := "PAR_SUB".FI_DIA_DYN_WIN_T1,       //filter time in sec.  
                tc_in          := 0.1,                             //interrupt time for filter module call (ts/tc>=1, ts/tc=integer!) 
                ts_in          := 0.1,                             //filter sample time
                max_delta      := 20.0,                            //default value for window increment after diameter mode is active
                min_delta      := 0.2,                             //min value for window increment
                rr             := "PAR_SUB".FI_DIA_DYN_WIN_RR / 10,  //parameter reject ratio
                i_count        := #count,                           //status buffer counter variable
                i_cycle        := #cycle,                           //status buffer cycle variable
                range_in       := "CNF".XT_DIA_RANGE,                //value for 100% input (e.g. 250mm = 100%) used for u_in   
                range_out      := "CNF".XT_DIA_RANGE,                //value for 100% output (e.g. 250mm = 100%) used for y_out
                y_llim         := 0.0,                             //low limit for y_out 
                y_hlim         := "CNF".XT_DIA_RANGE,                //high limit for y_out
                delta          := #delta_prev_call,                 //last window increment
                u_avg          := #dia_prev_call,                   //last valid diameter input
                y_out          := "AV".OUTP_XT_DIA_FIL);             //filter output

       //read filter times regarding running phase
       //-----------------------------------------
       IF "APC".STATUS = "APC".NECK THEN      
           "AC".CTL_DIA_TF_1 := "PAR_SUB".FI_DIA_NE_T1;                
           "AC".CTL_DIA_TF_2 := "PAR_SUB".FI_DIA_NE_T2;                
       ELSIF "APC".STATUS = "APC".SHOULDER THEN
           "AC".CTL_DIA_TF_1 := "PAR_SUB".FI_DIA_SH_T1;
           "AC".CTL_DIA_TF_2 := "PAR_SUB".FI_DIA_SH_T2;
       ELSE
           "AC".CTL_DIA_TF_1 := "PAR_SUB".FI_DIA_BY_T1;
           "AC".CTL_DIA_TF_2 := "PAR_SUB".FI_DIA_BY_T2;
       END_IF;

       //call PT2 filter
       //---------------
       #PT2 (u_in      := "AV".OUTP_XT_DIA_FIL,                    //filtered diameter input                      
            t1_in     := "AC".CTL_DIA_TF_1, 
            t2_in     := "AC".CTL_DIA_TF_2,
            ts_in     := 0.1,
            tc_in     := 0.1,
            range_in  := "CNF".XT_DIA_RANGE,
            range_out := "CNF".XT_DIA_RANGE,
            y_llim    := 0.0,
            y_hlim    := "CNF".XT_DIA_RANGE,
            y_out     := "AV".AVG_XT_DIA);  

       //select source of filtered diameter signal - added for usage of stereo camera
       //----------------------------------------------------------------------------
       IF (("CNF".ACT_DVC_CNF AND 2#0000_0000_0000_1000_0000_0000_0000_0000) = 2#0000_0000_0000_1000_0000_0000_0000_0000) THEN    
           "AV".ACT_XT_DIA       :=  "AV".S_CAM_AVG_XT_DIA;    //write diameter signal from stereo cameras
       ELSE
           "AV".ACT_XT_DIA       :=  "AV".AVG_XT_DIA;          //write diameter signal from single camera  
       END_IF;

       //write filtered actual value to display variable     
       //-----------------------------------------------
       #act             := "AV".ACT_XT_DIA;                                               
       "DIS".ACT_XT_DIA  := "AV".ACT_XT_DIA;

       //built controller on flag
       //------------------------
       IF "APC".AUTOMATIC AND NOT "SY".CTL_DIA_SMI AND NOT #ne_dia_ctrl_off THEN 
           "SY".CTL_DIA_ON := "DC".CTL_DIA_ON;  
       ELSE 
           "SY".CTL_DIA_ON := false; 
       END_IF;

       "LT".CTL_DIA_ON := "SY".CTL_DIA_ON;                             

       //diameter controller setpoint ramp
       //---------------------------------
       IF "SY".CTL_DIA_ON THEN                              
           //set crystal speed deviations
           //----------------------------
           IF ("SY".CTL_OFFS_SPEED_ON OR ("CTL".SET_SPEED_OFFS <> 0.0)) THEN    //gap/offset speed control is on or output of offset speed controller in ramp down stage
               #ll := "AC".SET_AVG_SPD;       //limitation equal to set point - >> pull speed fixes
               #hl := "AC".SET_AVG_SPD;
           //limitations according recipe columns
           //------------------------------------
           ELSE
               #ll := "AC".SET_XT_SPD_DEV_2;
               #hl := "AC".SET_XT_SPD_DEV_1;
           END_IF;

           IF ("APC".STATUS = "APC".BODY) THEN     //set point ramp only in body phase 
               IF (#set <> #set_prv_cyc) THEN    //compare setpoint with setpoint of previous cycle
                   #ramp_enb := true;           //enable ramp when setpoint has changed
               END_IF;
               #set_prv_cyc :=  #set;        //store setpoint of current cycle

               // call diameter controller setpoint ramp function
               //------------------------------------------------
               IF ("PAR_SUB".DIA_RP_GRAD > 0.0)     THEN
                   "CM_SET_RAMP"(rp_enb      := #ramp_enb,
                               i           := #cyc_cnt,
                               max_dev     := "PAR_SUB".DIA_RP_MAX_DEV,
                               rp_start    := "PAR_SUB".DIA_RP_START,
                               rp_grad     := "PAR_SUB".DIA_RP_GRAD,
                               tme_base    := 60.0,
                               tc_in       := 0.1,
                               set_p       := #set,
                               act_v       := #act,
                               set_out     := #set_ramp);

                   #set     := #set_ramp; 
               END_IF;      
           END_IF;     
       ELSE              
           #ll := 0.0;
           #hl := "CNF".XT_LFT_RANGE;

           #ramp_enb  := true;     
           #cyc_cnt   := true;                
       END_IF;

       //write setpoint to display value
       //-------------------------------
       "DIS".SET_XT_DIA := #set;

       //change polarity of control values
       //---------------------------------
       #set := #set *(-1);                                                          
       #act := #act *(-1);                                               

       //switch off diameter controller
       //------------------------------ 
       IF NOT "SY".CTL_DIA_ON    THEN 
           #ctl_dia_on  :=  false;
       END_IF;

       //enable of single controller actions
       //----------------------------------- 
       IF ("AC".CTL_DIA_TI > 0.0)   THEN         //i- part
           #int_action_on   :=  true;
       ELSE
           #int_action_on   :=  false;
       END_IF;

       IF ("AC".CTL_DIA_TD > 0.0)   THEN         //d-part
           #der_action_on   :=  true;
       ELSE
           #der_action_on   :=  false;
       END_IF;

       //write internal hand value
       //-------------------------
       IF NOT("SY".CTL_DIA_ON AND NOT #ctl_dia_on) THEN 
           //internal hand value scaling when fast in auto mode is requested
           //---------------------------------------------------------------
           IF (#hand > "CNF".XT_LFT_RANGE) THEN 
               #hand_int := #hand / "CNF_XT_LFT_LZ950".RATIO_FST_NRM;
           ELSE 
               #hand_int := #hand;
           END_IF;
       END_IF;

       //call Standard PID controller 
       //----------------------------
       #STD_PID(COM_RST         :=  "KYD".DIA_CTRL_RST,                   //restart of controller, resets controller values
               MAN_ON          :=  NOT #ctl_dia_on,                     //switch controller on/off
               PVPER_ON        :=  false,                              //activate reading of peripherie value
               P_SEL           :=  true,                               //proportional action on
               I_SEL           :=  #int_action_on,                      //integral action on
               INT_HOLD        :=  #int_hold_req,                       //integral action hold
               I_ITL_ON        :=  false,                              //initialization of the integral action - set value of I_ITLVAL
               D_SEL           :=  #der_action_on,                      //derivative action on
               CYCLE           :=  T#100ms,                            //sample time
               SP_INT          :=  #set,                                //internal setpoint
               PV_IN           :=  #act,                                //process variable input
               PV_PER          :=  W#16#0000,                          //process variable peripherial input
               MAN             :=  #hand_int / "CNF".XT_LFT_RANGE * 100.0,//hand value as percentaged input
               GAIN            :=  "AC".CTL_DIA_GN,                      //controller gain
               TI              :=  DINT_TO_TIME(REAL_TO_DINT("AC".CTL_DIA_TI * 1000.0)), //integration time
               TD              :=  DINT_TO_TIME(REAL_TO_DINT("AC".CTL_DIA_TD * 1000.0)), //derivative time
               TM_LAG          :=  DINT_TO_TIME(REAL_TO_DINT("AC".CTL_DIA_T1 * 1000.0)), //time lag of the derivative action
               DEADB_W         :=  0.0,                            //dead band of control deviation
               LMN_HLM         :=  #hl / "CNF".XT_LFT_RANGE * 100.0,  //upper limit of controller output as percentaged value 
               LMN_LLM         :=  #ll / "CNF".XT_LFT_RANGE * 100.0,  //lower limit of controller output as percentaged value
               PV_FAC          :=  1.0,                            //process variable factor (used on peripherial input)
               PV_OFF          :=  0.0,                            //process variable offset
               LMN_FAC         :=  1.0,                            //output standardization(percentage to physical value)
               LMN_OFF         :=  0.0,                            //offset of output value
               I_ITLVAL        :=  0.0,                            //initialization value of the integral action
               DISV            :=  #nc);                            //disturbance variable

               //write output variables of PID controller
               //----------------------------------------
               "CTL".SET_XT_SPD  :=  #STD_PID.LMN / 100.0 * "CNF".XT_LFT_RANGE; //controller output variable as physical value

               #per_out         :=  #STD_PID.LMN_PER;                        //peripherial controller output variable
               #high_lim_active :=  #STD_PID.QLMN_HLM;                       //high limit of controller output is reached
               #low_lim_active  :=  #STD_PID.QLMN_LLM;                       //low limit of controller output is reached
               #p_part_out      :=  #STD_PID.LMN_P;                          //proportionality component
               #i_part_out      :=  #STD_PID.LMN_I;                          //integral component
               #d_part_out      :=  #STD_PID.LMN_D;                          //derivative component
               #eff_act_val     :=  #STD_PID.PV;                             //effective process variable 
               #error_sig       :=  #STD_PID.ER;                             //control deviation

       //write display values of controller parts
       //----------------------------------------        
       "DIS".DIA_CONT_P  :=  #p_part_out / 100.0 * "CNF".XT_LFT_RANGE;
       "DIS".DIA_CONT_I  :=  #i_part_out / 100.0 * "CNF".XT_LFT_RANGE; 
       "DIS".DIA_CONT_D  :=  #d_part_out / 100.0 * "CNF".XT_LFT_RANGE;

       //output scaling when fast in auto mode is requested
       //--------------------------------------------------
       IF (#hand > "CNF".XT_LFT_RANGE) THEN 
           "CTL".SET_XT_SPD  :=  "CTL".SET_XT_SPD * "CNF_XT_LFT_LZ950".RATIO_FST_NRM; 
       END_IF;

       //evaluate controller output limits
       //---------------------------------
       IF #high_lim_active XOR #low_lim_active   THEN                //check controller limits
           IF (#ctrl_calls > 50) THEN                                   
               IF #high_lim_active AND (#i_part_out > 0.0)   THEN 
                   #int_hold_req    :=  true;                       //set integral action on hold
               ELSIF #low_lim_active AND (#i_part_out < 0.0) THEN 
                   #int_hold_req    :=  true;                       //set integral action on hold
               ELSE 
                   #int_hold_req    :=  false;                      //reset integral action on hold
               END_IF;
           ELSE
               #ctrl_calls  :=  #ctrl_calls + 1;                     //count controller calls
           END_IF;
       ELSE
           #ctrl_calls      :=  0;                                  //reset controller call counts
           #int_hold_req    :=  false;                              //reset integral action hold request
       END_IF;

       //switch on diameter controller
       //------------------------------ 
       IF "SY".CTL_DIA_ON    THEN 
           #ctl_dia_on  :=  true;
       END_IF;
END_FUNCTION_BLOCK

FUNCTION_BLOCK "CM_LOOP_HTR_1"   // FB136, SCL
{ S7_Optimized_Access := 'FALSE' }
VERSION : 0.0
// --------------------------------------------------------------------------------
//     program     :    CM_LOOP_HTR_1
//     description :    heater 1 control loop 
//     name        :    K. Kalkowski
//     date        :    08.12.99 
//     
//     revision    :    call of CONT_C added as alternative
//     name        :    G. Eibelsh鋟ser
//     date        :    07.09.2007
//     
//     revision    :    
//     name        :    
//     date        :    
// 
//                     (c)PVA TePla AG
//     --------------------------------------------------------------------------------
   VAR
      STD_PID : CONT_C;   // standard Siemens controller algorithm
      PT1_SET : "CM_PT1";   // pt1 filter for average heater 1 temperature set point
      PT1_ACT : "CM_PT1";   // pt1 filter for actual heater 1 temperature
      INC_PWR : "CM_INC";   // increment function power
      INC_TMP : "CM_INC";   // increment function temperature
      stp_1nc : Bool;
      stp_2nc : Bool;
      stp_3nc : Bool;
      rstrt_1nc : Bool;
      rstrt_2nc : Bool;
      rstrt_3nc : Bool;
      y0_tmp : Bool;   // y0 mode flag for temperature increment function
      stop_2_req : Bool;
      stop_3_req : Bool;
      status_avg_spd : Bool;
      status_mlt_tmp : Bool;
      status_grw_rte : Bool;
      status_dia_tmp : Bool;
      status_stp_2 : Bool;
      status_stp_3 : Bool;
      rstrt_mgs : Bool;
      rstrt_dia_tmp : Bool;
      ramp_enb : Bool;
      cyc_cnt : Bool;
      int_hold_req : Bool;   // integral hold action request
      pyr_failed : Bool;   // pyrometer failed
      ctl_htr_1_on : Bool;
      stat_avg_xt_spd : Bool;
      stat_avg_gap_offs : Bool;
      ctrl_calls : Int;   // controller call counter
      i : Int;
      set : Real;   // internal set point
      act : Real;   // internal actual value
      hand_tmp : Real;   // internal hand value temperature
      hand_pwr : Real;   // internal hand value power
      set_ramp : Real;
      pyr_act_htr_1_tmp_prv : Real;
      y_dia_tmp : Real;
   END_VAR
   VAR_TEMP
      high_lim_active : Bool;   // high limit of controller output is reached
      low_lim_active : Bool;   // low limit of controller output is reached
      int_action_on : Bool;   // integral action on
      der_action_on : Bool;   // derivative action on
      per_out : Word;   // peripherial controller output variable
      p_part_out : Real;   // proportionality component
      i_part_out : Real;   // integral component
      d_part_out : Real;   // derivative component
      eff_act_val : Real;   // effective process variable
      error_sig : Real;   // control deviation
   END_VAR
   VAR CONSTANT
      nc : Real := 0.0;   // "not connected input"
   END_VAR
BEGIN

                                                            //build hand value temperature 
       #hand_tmp := "CM_INSELECT" (auto   := ("APC".AUTOMATIC AND NOT "SY".CTL_HTR_1_SMI),        
                                track  := false,
                                ac     := "AC".SET_HTR_1_TMP,                
                                kya    := "KYA".SET_HTR_1_TMP);    


       IF "APC".AUTOMATIC    THEN
           IF "DC".CTL_PULL_RTE_ON  THEN              //select increment input from mgs control    
               IF "SY".CTL_AVG_CRUC_ROT_ON   THEN
                   "CTL".SET_HTR_1_MGS_INC := "CTL".Y_AVG_CRUC_ROT;        
               ELSE
                   //gap offset speed/gap control is used
                   //------------------------------------
                   IF "SY".CTL_OFFS_SPEED_ON THEN
                       //set restart request when average speed control was active last cycle
                       //--------------------------------------------------------------------
                       IF #stat_avg_xt_spd THEN
                           #rstrt_mgs := true;
                       //write output of average gap offset controller to increment input
                       //---------------------------------------------------------------- 
                       ELSE
                           "CTL".SET_HTR_1_MGS_INC   :=  "CTL".Y_AVG_GAP_OFFS;
                       END_IF;
                       #stat_avg_xt_spd         :=  false;
                       #stat_avg_gap_offs       :=  true;
                   //crystal average speed control is used
                   //-------------------------------------
                   ELSE
                       //set restart request when offset speed/gap control was active last cycle
                       //-----------------------------------------------------------------------
                       IF #stat_avg_gap_offs THEN
                           #rstrt_mgs := true; 
                       //write output of average pull speed controller to increment input
                       //---------------------------------------------------------------- 
                       ELSE
                           "CTL".SET_HTR_1_MGS_INC   :=  "CTL".Y_AVG_XT_SPD;
                       END_IF;
                       #stat_avg_xt_spd         :=  true;
                       #stat_avg_gap_offs       :=  false;
                   END_IF;
               END_IF;    
               IF #status_avg_spd = false THEN
                   #rstrt_mgs := true;
               END_IF;         
               #status_avg_spd := true;
               #status_mlt_tmp := false;
               #status_grw_rte := false;
               #status_stp_2   := false;

           ELSIF "DC".CTL_MLT_1_TMP_ON   THEN
               "CTL".SET_HTR_1_MGS_INC := "CTL".Y_MLT_1_TMP; 
               IF #status_mlt_tmp = false THEN
                   #rstrt_mgs := true;
               END_IF;         
               #status_avg_spd := false;
               #status_mlt_tmp := true;
               #status_grw_rte := false;
               #status_stp_2   := false;
               #stat_avg_xt_spd     :=  false;
               #stat_avg_gap_offs   :=  false;

           ELSIF "APC".AUTOMATIC AND "DC".CTL_GRW_RTE_ON   THEN 
               IF "SY".CTL_AVG_CRUC_ROT_ON   THEN
                   "CTL".SET_HTR_1_MGS_INC := "CTL".Y_AVG_CRUC_ROT;       
               ELSE
                   "CTL".SET_HTR_1_MGS_INC :=  "CTL".Y_GRW_RTE;
               END_IF;    
               IF #status_grw_rte = false THEN
                   #rstrt_mgs := true;
               END_IF;         
               #status_avg_spd := false;
               #status_mlt_tmp := false;
               #status_grw_rte := true;
               #status_stp_2   := false;
               #stat_avg_xt_spd     :=  false;
               #stat_avg_gap_offs   :=  false;

           ELSE
               "CTL".SET_HTR_1_MGS_INC := 0.0;
               #status_avg_spd := false;
               #status_mlt_tmp := false;
               #status_grw_rte := false;
               #stat_avg_xt_spd     :=  false;
               #stat_avg_gap_offs   :=  false;

               IF #status_stp_2 = false THEN
                   #stop_2_req := true;
               END_IF;
               #status_stp_2 := true;
           END_IF;    
       ELSE
           "CTL".SET_HTR_1_MGS_INC := 0.0;
           #status_avg_spd := false;
           #status_mlt_tmp := false;
           #status_grw_rte := false;

           IF #status_stp_2 = false THEN
               #stop_2_req := true;
           END_IF;
           #status_stp_2 := true;
       END_IF;

       //increment input 3
       //-----------------
       IF "DC".CTL_DIA_ON THEN                                       //diameter control is requested
           //write output of diameter- temperature controller
           //------------------------------------------------
           #y_dia_tmp   := "CTL".Y_DIA_TMP; 
           //write control bits of inc input 3
           //---------------------------------
           IF NOT #status_dia_tmp THEN
               #rstrt_dia_tmp := true;
           END_IF;         
           #status_dia_tmp := true;
           #status_stp_3   := false;
       ELSE                                                        //diameter control is not requested
           //write output of diameter- temperature controller
           //------------------------------------------------
           #y_dia_tmp   := 0.0; 
           //write control bits of inc input 3
           //---------------------------------
           #status_dia_tmp := false;
           IF NOT #status_stp_3 THEN
               #stop_3_req := true;
           END_IF;
           #status_stp_3 := true;
       END_IF;

       IF "APC".AUTOMATIC AND NOT "SY".CTL_HTR_1_SMI THEN      //y0_mode condition for temperature increment 
           #y0_tmp := "DC".SET_HTR_1_TMP_ABS;
       ELSE
           #y0_tmp := true;
       END_IF;

       #INC_TMP (u1_in       := "AC".SET_HTR_1_TMP_INC,       //build set point temperature           
                u2_in       := "CTL".SET_HTR_1_MGS_INC,            
                u3_in       := #y_dia_tmp,                  //input from diameter- temperature controller            
                k1_in       := 1.0,
                k2_in       := 1.0,
                k3_in       := 1.0,
                y0_in       := #hand_tmp,
                y_llim      := "CNF".HTR_1_TMP_RANGE_LOW, 
                y_hlim      := "CNF".HTR_1_TMP_RANGE_HI,
                y0_mode     := #y0_tmp,                       
                y_out       := "CTL".SET_HTR_1_TMP,
                stp_1       := #stp_1nc,                       
                stp_2       := #stop_2_req,
                stp_3       := #stop_3_req,
                rstrt_1     := "DC".RSTRT_HTR_1_TMP_INC,    
                rstrt_2     := #rstrt_mgs,
                rstrt_3     := #rstrt_dia_tmp);
       #set:= "CTL".SET_HTR_1_TMP;

       //display heater 1 temperature increment related to start of phase
       //----------------------------------------------------------------
       IF (("APC".STATUS >= "APC".NECK) AND ("APC".STATUS <= "APC".ENDCONE))  THEN  
           IF ("STA".ACT_STE_NO > 100) THEN  //process phase is running
               "DIS".ACT_HTR_1_TMP_INC   :=  "CTL".SET_HTR_1_TMP - "DIS".HTR_1_TMP_SET_PHA_STR;
           END_IF;

           "DIS".SET_HTR_1_TMP_INC   :=  "AC".SET_HTR_1_TMP_INC;   //write recipe value to actual heater 1 increment variable

       ELSE
           "DIS".ACT_HTR_1_TMP_INC   :=  0.0;
           "DIS".SET_HTR_1_TMP_INC   :=  0.0;
       END_IF;


       "AC".CTL_HTR_1_AVG_TMP_TF := "PAR_SUB".FI_AV_TMP_1;    //fetch filter time from PAR_SUB db  
       "AC".CTL_HTR_1_TMP_TF := "PAR_SUB".FI_TMP_HTR_1; 


       #PT1_SET (u_in      := "CTL".SET_HTR_1_TMP,            //build average heater temperature set point                      
                t1_in     := "AC".CTL_HTR_1_AVG_TMP_TF, 
                ts_in     := 0.1,
                tc_in     := 0.1,
                range_in  := "CNF".HTR_1_TMP_RANGE_HI,
                range_out := "CNF".HTR_1_TMP_RANGE_HI,
                y_llim    := "CNF".HTR_1_TMP_RANGE_LOW,
                y_hlim    := "CNF".HTR_1_TMP_RANGE_HI,
                y_out     := "AV".AVG_HTR_1_TMP);            //only display value, no control function

       "DIS".ACT_HTR_1_AV_TMP := "AV".AVG_HTR_1_TMP;            //set display values
       "DIS".SET_HTR_1_PWR := "CTL".SET_HTR_1_PWR;

       #PT1_ACT (u_in      := "PAI".PYR_ACT_HTR_1_TMP,         //build actual temperature value temperature                      
                t1_in     := "AC".CTL_HTR_1_TMP_TF, 
                ts_in     := 0.1,
                tc_in     := 0.1,
                range_in  := "CNF".HTR_1_TMP_RANGE_HI,
                range_out := "CNF".HTR_1_TMP_RANGE_HI,
                y_llim    := "CNF".HTR_1_TMP_RANGE_LOW,
                y_hlim    := "CNF".HTR_1_TMP_RANGE_HI,
                y_out     := "AV".ACT_HTR_1_TMP); 

       #act := "AV".ACT_HTR_1_TMP;                                               

       "DIS".ACT_HTR_1_TMP := "AV".ACT_HTR_1_TMP;

       //check pyrometer signal when temperature control is on
       //-----------------------------------------------------
       IF "SY".CTL_HTR_1_ON  THEN
           //calculate deviation of temperature from last cycle
           //--------------------------------------------------
           IF ((#pyr_act_htr_1_tmp_prv - "PAI".PYR_ACT_HTR_1_TMP) > 15.0) THEN  //temp. drop larger 15癈
               #pyr_failed  :=  true;
           END_IF;

       ELSE
           //reset signal "pyrometer failed" with delay
           //------------------------------------------
           IF #pyr_failed   THEN 
               IF (#i > 50)    THEN             //delay reset at least 5 seconds
                   IF NOT "APC".AUTOMATIC THEN
                       #pyr_failed  :=  false;  //reset failure flag when automatic is off
                   END_IF;
               ELSE 
                   #i   :=  #i + 1;  //increment 100ms counter
               END_IF; 
           ELSE 
               #i   :=  0;  //reset counter value
           END_IF;

       END_IF; 

       //store actual temperature for one 100ms cycle
       //--------------------------------------------
       #pyr_act_htr_1_tmp_prv   :=  "PAI".PYR_ACT_HTR_1_TMP;    

       //set fault message when pyrometer failed
       //---------------------------------------
       "FLT".HTR_1_TMP_SIG   :=  #pyr_failed;

       //switch temperature control on/off
       //---------------------------------
       IF "LT".HTR_1_ON AND NOT #pyr_failed THEN

           IF "APC".AUTOMATIC AND NOT "SY".CTL_HTR_1_SMI THEN    //build control on flag
               "SY".CTL_HTR_1_ON := "DC".CTL_HTR_1_TMP_ON;                 
           ELSE 
               "SY".CTL_HTR_1_ON := ("SY".CTL_HTR_1_ON AND NOT "KYD".CTL_HTR_1_TMP_OFF) OR "KYD".CTL_HTR_1_TMP_ON; 
           END_IF;

       ELSE
           "SY".CTL_HTR_1_ON := false;

       END_IF;

       // call setpoint ramp function after controller start
       //---------------------------------------------------
       IF "SY".CTL_HTR_1_ON  THEN
           IF ("PAR_SUB".HTR_1_TMP_RP_GRAD > 0.0)     THEN
               "CM_SET_RAMP"(rp_enb      := #ramp_enb,
                           i           := #cyc_cnt,
                           max_dev     := "PAR_SUB".HTR_1_TMP_RP_MAX_DEV,
                           rp_start    := "PAR_SUB".HTR_1_TMP_RP_START,
                           rp_grad     := "PAR_SUB".HTR_1_TMP_RP_GRAD,
                           tme_base    := 60.0,
                           tc_in       := 0.1,
                           set_p       := #set,
                           act_v       := #act,
                           set_out     := #set_ramp);

               #set     := #set_ramp; 
           END_IF;
       ELSE
           #ramp_enb  := TRUE;     
           #cyc_cnt   := TRUE;                
       END_IF;

       //display heater temperature setpoint
       //-----------------------------------
       "DIS".SET_HTR_1_TMP := #set;

       //track manual setpoint when control is off
       //-----------------------------------------
       IF NOT "SY".CTL_HTR_1_ON  THEN                        
           "KYA".SET_HTR_1_TMP   :=  "AV".ACT_HTR_1_TMP;   //manual setpoint variable tracked with actual value

       //track manual setpoint when control is on
       //----------------------------------------
       ELSIF "APC".AUTOMATIC AND NOT "SY".CTL_HTR_1_SMI THEN   //manual setpoint variable tracked with actual setpoint
           "KYA".SET_HTR_1_TMP := #set;
       END_IF;                                                         

       "LT".CTL_HTR_1_TMP_ON := "SY".CTL_HTR_1_ON;                             

       //write PID parameters of heater temperature control phase related
       //----------------------------------------------------------------
       IF ("APC".STATUS = "APC".DIPPING)   THEN          
           "AC".CTL_HTR_1_TMP_GN := "PAR_MAIN".CTL_HTR_1_TMP_GN_DIP;
           "AC".CTL_HTR_1_TMP_TI := "PAR_MAIN".CTL_HTR_1_TMP_TI_DIP;
           "AC".CTL_HTR_1_TMP_TD := "PAR_MAIN".CTL_HTR_1_TMP_TD_DIP;
           "AC".CTL_HTR_1_TMP_T1 := "PAR_MAIN".CTL_HTR_1_TMP_T1_DIP;

       ELSE
           "AC".CTL_HTR_1_TMP_GN := "PAR_MAIN".CTL_HTR_1_TMP_GN;
           "AC".CTL_HTR_1_TMP_TI := "PAR_MAIN".CTL_HTR_1_TMP_TI;
           "AC".CTL_HTR_1_TMP_TD := "PAR_MAIN".CTL_HTR_1_TMP_TD;
           "AC".CTL_HTR_1_TMP_T1 := "PAR_MAIN".CTL_HTR_1_TMP_T1;
       END_IF;

       //do controller call
       //------------------

           //switch off heater temperature controller
           //---------------------------------------- 
           IF NOT "SY".CTL_HTR_1_ON    THEN 
               #ctl_htr_1_on  :=  false;
           END_IF;

           //enable of single controller actions
           //----------------------------------- 
           IF ("AC".CTL_HTR_1_TMP_TI > 0.0)   THEN         //i- part
               #int_action_on   :=  true;
           ELSE
               #int_action_on   :=  false;
           END_IF;

           IF ("AC".CTL_HTR_1_TMP_TD > 0.0)   THEN         //d-part
               #der_action_on   :=  true;
           ELSE
               #der_action_on   :=  false;
           END_IF;

           //call Standard PID controller 
           //----------------------------
           #STD_PID(COM_RST         :=  "KYD".HTR_1_CTRL_RST,                 //restart of controller, resets controller values
                   MAN_ON          :=  NOT #ctl_htr_1_on,                   //switch controller on/off
                   PVPER_ON        :=  false,                              //activate reading of peripherie value
                   P_SEL           :=  true,                               //proportional action on
                   I_SEL           :=  #int_action_on,                      //integral action on
                   INT_HOLD        :=  #int_hold_req,                       //integral action hold
                   I_ITL_ON        :=  false,                              //initialization of the integral action - set value of I_ITLVAL
                   D_SEL           :=  #der_action_on,                      //derivative action on
                   CYCLE           :=  T#100ms,                            //sample time
                   SP_INT          :=  #set,                                //internal setpoint
                   PV_IN           :=  #act,                                //process variable input
                   PV_PER          :=  W#16#0000,                          //process variable peripherial input
                   MAN             :=  0.0,                                //hand value as percentaged input
                   GAIN            :=  "AC".CTL_HTR_1_TMP_GN,                //controller gain
                   TI              :=  DINT_TO_TIME(REAL_TO_DINT("AC".CTL_HTR_1_TMP_TI * 1000.0)),   //integration time
                   TD              :=  DINT_TO_TIME(REAL_TO_DINT("AC".CTL_HTR_1_TMP_TD * 1000.0)),   //derivative time
                   TM_LAG          :=  DINT_TO_TIME(REAL_TO_DINT("AC".CTL_HTR_1_TMP_T1 * 1000.0)),   //time lag of the derivative action
                   DEADB_W         :=  0.0,                            //dead band of control deviation
                   LMN_HLM         :=  100.0,                          //upper limit of controller output as percentaged value 
                   LMN_LLM         :=  -100.0,                         //lower limit of controller output as percentaged value
                   PV_FAC          :=  1.0,                            //process variable factor (used on peripherial input)
                   PV_OFF          :=  0.0,                            //process variable offset
                   LMN_FAC         :=  1.0,                            //output standardization(percentage to physical value)
                   LMN_OFF         :=  0.0,                            //offset of output value
                   I_ITLVAL        :=  0.0,                            //initialization value of the integral action
                   DISV            :=  #nc);                            //disturbance variable

                   //write output variables of PID controller
                   //----------------------------------------
                   "CTL".SET_HTR_1_PWR_INC   :=  #STD_PID.LMN / 100.0 * "CNF".HTR_1_PWR_RANGE;  //controller output variable as physical value

                   #per_out         :=  #STD_PID.LMN_PER;                    //peripherial controller output variable
                   #high_lim_active :=  #STD_PID.QLMN_HLM;                   //high limit of controller output is reached
                   #low_lim_active  :=  #STD_PID.QLMN_LLM;                   //low limit of controller output is reached
                   #p_part_out      :=  #STD_PID.LMN_P;                      //proportionality component
                   #i_part_out      :=  #STD_PID.LMN_I;                      //integral component
                   #d_part_out      :=  #STD_PID.LMN_D;                      //derivative component
                   #eff_act_val     :=  #STD_PID.PV;                         //effective process variable 
                   #error_sig       :=  #STD_PID.ER;                         //control deviation

           //write display values of controller parts
           //----------------------------------------        
           "DIS".HTR_1_CONT_P    :=  #p_part_out / 100.0 * "CNF".HTR_1_PWR_RANGE; 
           "DIS".HTR_1_CONT_I    :=  #i_part_out / 100.0 * "CNF".HTR_1_PWR_RANGE; 
           "DIS".HTR_1_CONT_D    :=  #d_part_out / 100.0 * "CNF".HTR_1_PWR_RANGE; 

           //evaluate controller output limits
           //---------------------------------
           IF #high_lim_active XOR #low_lim_active   THEN                //check controller limits
               IF (#ctrl_calls > 50) THEN                                   
                   IF #high_lim_active AND (#i_part_out > 0.0)   THEN 
                       #int_hold_req    :=  true;                       //set integral action on hold
                   ELSIF #low_lim_active AND (#i_part_out < 0.0) THEN 
                       #int_hold_req    :=  true;                       //set integral action on hold
                   ELSE 
                       #int_hold_req    :=  false;                      //reset integral action on hold
                   END_IF;
               ELSE
                   #ctrl_calls  :=  #ctrl_calls + 1;                     //count controller calls
               END_IF;
           ELSE
               #ctrl_calls      :=  0;                                  //reset controller call counts
               #int_hold_req    :=  false;                              //reset integral action hold request
           END_IF;

           //switch on heater temperature controller
           //--------------------------------------- 
           IF "SY".CTL_HTR_1_ON    THEN 
               #ctl_htr_1_on  :=  true;
           END_IF;

       //build hand value power
       //----------------------
       #hand_pwr := "CM_INSELECT" (auto   := ("APC".AUTOMATIC AND NOT "SY".CTL_HTR_1_SMI),        
                                track  := false,
                                ac     := "AC".SET_HTR_1_PWR,                
                                kya    := "KYA".SET_HTR_1_PWR);   

       //call increment function and built power setpoint
       //------------------------------------------------
       #INC_PWR (u1_in       := "CTL".SET_HTR_1_PWR_INC,            
                u2_in       := 0.0,            
                u3_in       := 0.0,            
                k1_in       := 1.0,
                k2_in       := 0.0,
                k3_in       := 0.0,
                y0_in       := #hand_pwr,
                y_llim      := 0.0, 
                y_hlim      := "CNF".HTR_1_PWR_RANGE,
                y0_mode     := NOT "SY".CTL_HTR_1_ON,                       
                y_out       := "CTL".SET_HTR_1_PWR,
                stp_1       := #stp_1nc,                       
                stp_2       := #stp_2nc,
                stp_3       := #stp_3nc,
                rstrt_1     := #rstrt_1nc,    
                rstrt_2     := #rstrt_2nc,
                rstrt_3     := #rstrt_3nc);

       //track hand power setpoint while automatic or temperature control is active 
       //--------------------------------------------------------------------------
       IF ("APC".AUTOMATIC AND NOT "SY".CTL_HTR_1_SMI) OR "SY".CTL_HTR_1_ON THEN    
           IF "SY".CTL_HTR_1_ON THEN 
               "KYA".SET_HTR_1_PWR := "CTL".SET_HTR_1_PWR;
           ELSIF  ("APC".STATUS = "APC".MELTING OR "APC".STATUS = "APC".DIPPING OR "APC".STATUS = "APC".SHUT_DOWN) THEN  
               "KYA".SET_HTR_1_PWR := "AC".SET_HTR_1_PWR;
           END_IF;
      END_IF;
END_FUNCTION_BLOCK

FUNCTION_BLOCK "CM_LOOP_HTR_2"   // FB137, SCL
{ S7_Optimized_Access := 'FALSE' }
VERSION : 0.0
// --------------------------------------------------------------------------------
//     program     :    CM_LOOP_HTR_2
//     description :    heater 2 control loop 
//     name        :    K. Kalkowski
//     date        :    10.12.99 
// 
//     revision    :    
//     name        :    
//     date        :    
// 
//                     (c)PVA TePla AG
//     --------------------------------------------------------------------------------
   VAR
      PT1 : "CM_PT1";   // pt1 filter for heater 2 temperature
      INC : "CM_INC";   // increment function power
      hand : Real;   // internal hand value
      y0 : Bool;   // y0 condition for power inc
      nc : Real;   // "not connected" input
      stp_1nc : Bool;
      stp_2nc : Bool;
      stp_3nc : Bool;
      rstrt_1nc : Bool;
      rstrt_2nc : Bool;
      rstrt_3nc : Bool;
   END_VAR
BEGIN

                                                       //build hand value 
       #hand := "CM_INSELECT" (auto   := ("APC".AUTOMATIC AND NOT "SY".CTL_HTR_2_SMI),        
                            track  := false,
                            ac     := "AC".SET_HTR_2_PWR,                
                            kya    := "KYA".SET_HTR_2_PWR);  


     //  PT1     (u_in      := PAI.PYR_ACT_HTR_2_TMP,        //build actual temperature value temperature                      
     //           t1_in     := AC.CTL_HTR_2_TMP_TF, 
     //           ts_in     := 0.1,
     //           tc_in     := 0.1,
     //           range_in  := CNF.HTR_2_TMP_RANGE_HI,
     //           range_out := CNF.HTR_2_TMP_RANGE_HI,
     //           y_llim    := CNF.HTR_2_TMP_RANGE_LOW,
     //           y_hlim    := CNF.HTR_2_TMP_RANGE_HI,
     //           y_out     := AV.ACT_HTR_2_TMP); 


       IF "APC".AUTOMATIC AND NOT "SY".CTL_HTR_2_SMI THEN      //y0_mode condition for power increment 
           #y0 := "DC".SET_HTR_2_PWR_ABS;
       ELSE
           #y0 := true;
       END_IF;

       //call increment function
       //-----------------------
       #INC     (u1_in       := "AC".SET_HTR_2_PWR_INC,      //build set point power           
                u2_in       := "CTL".SET_HTR_1_PWR,            
                u3_in       := 0.0,            
                k1_in       := 1.0,
                k2_in       := "AC".PWR_COEFF_2 / 100,    
                k3_in       := 0.0,
                y0_in       := #hand,
                y_llim      := 0.0, 
                y_hlim      := "CNF".HTR_2_PWR_RANGE,
                y0_mode     := #y0,                       
                y_out       := "CTL".SET_HTR_2_PWR,
                stp_1       := #stp_1nc,                       
                stp_2       := #stp_2nc,
                stp_3       := #stp_3nc,
                rstrt_1     := "DC".RSTRT_HTR_2_PWR_INC,    
                rstrt_2     := #rstrt_2nc,
                rstrt_3     := #rstrt_3nc);

       IF "APC".AUTOMATIC AND NOT "SY".CTL_HTR_2_SMI THEN      //track hand power set point
           "KYA".SET_HTR_2_PWR := "CTL".SET_HTR_2_PWR;
       END_IF;                                                         

       "DIS".SET_HTR_2_PWR := "CTL".SET_HTR_2_PWR;             //set display value

       //display heater 2 power increment related to start of phase
       //----------------------------------------------------------
       IF (("APC".STATUS >= "APC".NECK) AND ("APC".STATUS <= "APC".ENDCONE))  THEN  
           "DIS".SET_HTR_2_PWR_INC   :=  "AC".SET_HTR_2_PWR_INC + "CTL".SET_HTR_1_PWR * "AC".PWR_COEFF_2 / 100;
       ELSE
           "DIS".SET_HTR_2_PWR_INC   :=  0.0;
       END_IF;
END_FUNCTION_BLOCK

FUNCTION_BLOCK "CM_LOOP_AVG_SPD"   // FB138, SCL
{ S7_Optimized_Access := 'FALSE' }
VERSION : 0.0
// --------------------------------------------------------------------------------
//     program     :    CM_LOOP_AVG_SPD
//     description :    average speed control loop 
//     name        :    K. Kalkowski
//     date        :    11.12.99 
// 
//     revision    :    call of CONT_C added as alternative
//     name        :    G. Eibelsh鋟ser
//     date        :    07.09.2007
//     
//     revision    :    
//     name        :    
//     date        :    
// 
//                     (c)PVA TePla AG
//     --------------------------------------------------------------------------------
   VAR
      STD_PID : CONT_C;   // standard Siemens controller algorithm
      PT1 : "CM_PT1";   // pt1 filter for average xtal speed
      ramp_enb : Bool;
      cyc_cnt : Bool;
      int_hold_req : Bool;   // integral hold action request
      ctl_avg_spd_on : Bool;
      ctrl_calls : Int;   // controller call counter
      set : Real;   // internal set point
      act : Real;   // internal actual value
      hand : Real;   // internal hand value
      ll : Real;   // controller output low limit
      hl : Real;   // controller output high limit
      ro : Real;   // controller output range
      set_ramp : Real;
      z_input : Real;   // interference input
      z_input_old : Real;   // interference input of previous cycle
      set_avg_cruc_rot_old : Real;   // average crucible rotation setpoint of previous cycle
   END_VAR
   VAR_TEMP
      high_lim_active : Bool;   // high limit of controller output is reached
      low_lim_active : Bool;   // low limit of controller output is reached
      int_action_on : Bool;   // integral action on
      der_action_on : Bool;   // derivative action on
      per_out : Word;   // peripherial controller output variable
      p_part_out : Real;   // proportionality component
      i_part_out : Real;   // integral component
      d_part_out : Real;   // derivative component
      eff_act_val : Real;   // effective process variable
      error_sig : Real;   // control deviation
   END_VAR
   VAR CONSTANT
      nc : Real := 0.0;   // "not connected" input
   END_VAR
BEGIN

        //built hand value
       //----------------
       IF ("PAR_MAIN".BY_CRUC_ROT_CTL_ON = 1.0) THEN       //average crucible rotation control is active
           IF   ("APC".STATUS <> "APC".SHOULDER)   THEN      //shoulder mode not running

               //built hand value of crucible rotation setpoint
               //----------------------------------------------
               IF  "APC".AUTOMATIC AND NOT "SY".CTL_CR_ROT_SMI AND "DV".TRANS_SH_BY_FLAG    THEN 
                   #hand    := "CTL".SET_CR_ROT; //keep last setpoint from shoulder as setpoint for body start  
               ELSE
                   #hand    := "CM_INSELECT" (auto  := ("APC".AUTOMATIC AND NOT "SY".CTL_CR_ROT_SMI),        
                                           track  := false,
                                           ac     := "AC".SET_CR_ROT,                
                                           kya    := "KYA".SET_CR_ROT);
               END_IF;

               //transform to percentage value
               //-----------------------------
               IF "DV".SPD_CTRL_STD_ALG    THEN    //only when standard PID algorithm is active
                   #hand := #hand / "CNF".CR_ROT_RANGE * 100.0;
               END_IF;

           END_IF;

       ELSE                    //average crucible rotation control is passive
           #hand := 0.0;        //no hand value 

       END_IF;   

       //read setpoint form recipe
       //-------------------------                                                    
       #set := "AC".SET_AVG_SPD;               

       //read filter time from recipe 
       //----------------------------
       "AC".CTL_AV_SPD_TF := "PAR_SUB".FI_AV_SPD;

       //call filter algorithm and built average crystal speed actual value 
       //------------------------------------------------------------------   
       #PT1 (u_in      := "CTL".SET_XT_SPD,                          
            t1_in     := "AC".CTL_AV_SPD_TF, 
            ts_in     := 0.1,
            tc_in     := 0.1,
            range_in  := "CNF".XT_LFT_RANGE,
            range_out := "CNF".XT_LFT_RANGE,
            y_llim    := 0.0,
            y_hlim    := "CNF".XT_LFT_RANGE,
            y_out     := "CTL".AVG_XT_SPD); 

       "DIS".ACT_XT_AV_SPD   := "CTL".AVG_XT_SPD;
       #act                 := "CTL".AVG_XT_SPD;    

       //build controller on flag
       //------------------------                                           
       IF "APC".AUTOMATIC AND NOT "SY".CTL_HTR_1_SMI THEN                               
           IF "SY".CTL_AVG_CRUC_ROT_ON   THEN
               IF  NOT "SY".CTL_CR_ROT_SMI   THEN
                   "SY".CTL_AVG_SPD_ON := "DC".CTL_PULL_RTE_ON;    //set flag according to process mode                 
               ELSE 
                   "SY".CTL_AVG_SPD_ON := FALSE;                 //switch off if cruc rot is in semi mode
               END_IF;
           ELSE    
               "SY".CTL_AVG_SPD_ON := "DC".CTL_PULL_RTE_ON;        //set flag according to process mode
           END_IF;
       ELSE
           "SY".CTL_AVG_SPD_ON := FALSE;                         //switch off pull rate control in manuell mode
       END_IF;        

       "LT".CTL_AV_SPD_ON := "SY".CTL_AVG_SPD_ON;                  //set light variable if pull rate control is on

       //check process mode and controller output range
       //----------------------------------------------
       IF ("APC".STATUS = "APC".BODY) AND ("PAR_MAIN".BY_CRUC_ROT_CTL_ON = 1.0)  THEN
           IF "SY".CTL_AVG_SPD_ON    THEN
               IF "DV".SPD_CTRL_STD_ALG  THEN 
                   #ll  :=  "AC".SET_CRUC_ROT_DEV_2 / "CNF".CR_ROT_RANGE * 100.0;
                   #hl  :=  "AC".SET_CRUC_ROT_DEV_1 / "CNF".CR_ROT_RANGE * 100.0;
                   #ro  :=  "CNF".CR_ROT_RANGE / 100.0;
               ELSE
                   #ll  :=  "AC".SET_CRUC_ROT_DEV_2;
                   #hl  :=  "AC".SET_CRUC_ROT_DEV_1;
                   #ro  :=  "CNF".CR_ROT_RANGE;
               END_IF;

           ELSE
               IF "DV".SPD_CTRL_STD_ALG  THEN 
                   #ll  :=  0.0;
                   #hl  :=  100.0;
                   #ro  :=  "CNF".CR_ROT_RANGE / 100.0;
               ELSE
                   #ll  :=  0.0;
                   #hl  :=  "CNF".CR_ROT_RANGE;
                   #ro  :=  "CNF".CR_ROT_RANGE;
               END_IF;
           END_IF;      
       ELSE
           IF "DV".SPD_CTRL_STD_ALG  THEN 
               #ll  :=  -100.0;
               #hl  :=  100.0;
               #ro  :=  "CNF".HTR_1_TMP_RANGE_HI / 100.0;
           ELSE
               #ll  :=  "CNF".HTR_1_TMP_RANGE_HI *(-1);
               #hl  :=  "CNF".HTR_1_TMP_RANGE_HI;
               #ro  :=  "CNF".HTR_1_TMP_RANGE_HI;
           END_IF;
       END_IF;

       IF "SY".CTL_AVG_SPD_ON  THEN
           // call setpoint ramp function after controller start
           //---------------------------------------------------
           IF ("PAR_SUB".AV_PULL_SPD_RP_GRAD > 0.0)     THEN
               "CM_SET_RAMP"(rp_enb      := #ramp_enb,
                           i           := #cyc_cnt,
                           max_dev     := "PAR_SUB".AV_PULL_SPD_RP_MAX_DEV,
                           rp_start    := "PAR_SUB".AV_PULL_SPD_RP_START,
                           rp_grad     := "PAR_SUB".AV_PULL_SPD_RP_GRAD,
                           tme_base    := 60.0,
                           tc_in       := 0.1,
                           set_p       := #set,
                           act_v       := #act,
                           set_out     := #set_ramp);

               #set     := #set_ramp; 
           END_IF;
       ELSE
           #ramp_enb  := TRUE;     
           #cyc_cnt   := TRUE;                
       END_IF;

       "DIS".SET_XT_AV_SPD := #set;

       //reset saved interference variables for cruc rot control if pull speed controller is off
       //---------------------------------------------------------------------------------------
       IF ("SY".CTL_AVG_SPD_ON = FALSE)  THEN
           #z_input_old          := 0.0;
           #set_avg_cruc_rot_old := "AC".SET_AVG_CRUC_ROT;
       END_IF;                            

       //change polarity of setpoint and actual if crucible rotation control is off
       //--------------------------------------------------------------------------
       IF ("PAR_MAIN".BY_CRUC_ROT_CTL_ON = 0.0) THEN
           #set     := #set *(-1);
           #act     := #act *(-1);
           #z_input := 0.0;             // keep interference input 0.0, if crucible rotation control is off

       //set interference input with average crucible rotation profile
       //-------------------------------------------------------------
       ELSE
           #z_input := #z_input_old + (#set_avg_cruc_rot_old - "AC".SET_AVG_CRUC_ROT) * (-1);   

           //transform to percentage value when standard algorithm is set
           //------------------------------------------------------------
           IF "DV".SPD_CTRL_STD_ALG  THEN
               #z_input := #z_input / "CNF".CR_ROT_RANGE * 100.0;
           END_IF;
       END_IF;    

       //do controller call
       //------------------

           //switch off average pull speed controller
           //---------------------------------------- 
           IF NOT "SY".CTL_AVG_SPD_ON    THEN 
               #ctl_avg_spd_on  :=  false;
           END_IF;

